FUNCTION_BLOCK FB_HMIConfigure EXTENDS FB_Base IMPLEMENTS ITF_HMIConfigure
VAR
	(*	Baza konfiguracji	*)
	arritfConfigure				: ARRAY [1..10] OF ITF_HMIConfiguration;
	iNubmerOfAddedConfigure		: INT;
END_VAR

METHOD PUBLIC AddConfiguration : BOOL
VAR_INPUT
	fbConfigure		: ITF_HMIConfiguration;
END_VAR
IF (THIS^.iNubmerOfAddedConfigure + 1 <= 10) THEN
	THIS^.iNubmerOfAddedConfigure	:= THIS^.iNubmerOfAddedConfigure + 1;
	THIS^.arritfConfigure [THIS^.iNubmerOfAddedConfigure]	:= fbConfigure;
	AddConfiguration	:= TRUE;
ELSE
	AddConfiguration	:= FALSE;
END_IF
END_METHOD

METHOD PUBLIC Configure : BOOL
VAR_INPUT
	fbHMIManager			: ITF_HMIManagerConfigure;
END_VAR
VAR
	bResult				: BOOL;
	iI					: INT;
END_VAR
bResult			:= TRUE;

THIS^.arritfConfigure [1].AddMainMenu (itfHMIManager := fbHMIManager);
THIS^.arritfConfigure [1].AddMachineControlConnector (itfHMIManager := fbHMIManager);
THIS^.arritfConfigure [1].AddPrepareScreenModule (itfHMIManager := fbHMIManager);

FOR iI := 1 TO THIS^.iNubmerOfAddedConfigure DO 
	IF (THIS^.arritfConfigure [iI] <> 0) THEN
		THIS^.arritfConfigure [iI].SetButtonActive (itfHMIManager	:= fbHMIManager);
		THIS^.arritfConfigure [iI].SetButtonsVisible (itfHMIManager	:= fbHMIManager);
		THIS^.arritfConfigure [iI].SetButtonsEnabled (itfHMIManager	:= fbHMIManager);
		//THIS^.arritfConfigure [iI].

	END_IF
END_FOR

THIS^.arritfConfigure [1].LinkHMIManagerData (itfHMIManager := fbHMIManager);

Configure		:= bResult;
END_METHOD

END_FUNCTION_BLOCK

(* stored: Version 1.1.0.1
   POU FB_HMIConfigure: Id {1396ad99-d92c-4ed4-a711-16f2a071df52}, SpecialFunc None
   Method AddConfiguration: Id {668b04e9-50eb-4ae1-9dd6-f7187fdbc317}
   Method Configure: Id {4a465225-aae0-41c8-ad3c-fe75dc47ce84} *)
